//{attribute 'qualified_only'}
VAR_GLOBAL

END_VAR

(* stored: Version 1.1.0.1, ProductVersion 3.1.4024.4
   GVL GVL_ActionModule: Id {713d5004-c073-4faa-a277-b1de756331a7} *)
